FUNCTION F_t_v0 : TIME
VAR_INPUT
	PosnDelta	: LREAL;
	Accel		: LREAL;
END_VAR
VAR
END_VAR

IF Accel <> 0 THEN
	F_t_v0	:= LREAL_TO_TIME(SQRT((2*PosnDelta)/Accel));
END_IF

END_FUNCTION

(* stored: Version 1.1.0.1
   POU F_t_v0: Id {44389f47-6186-02c6-24ef-53943624ab4b}, SpecialFunc None *)
